# EPICS substitutions: llrfHlsAsynApp/Db/llrfHlsAsyn.substitutions
file config.db
{
    pattern {   DEVICE,  NELM_BL, NELM_HARMO  }
            {  "$(DEV)",    4096,         18  }
}

file status.db
{
    pattern {   DEVICE,  NELM_ALPHA  }
             { "$(DEV)",          7  }
}

file config_ch.db
{
    pattern { CH,  DEVICE   }
            {  0,  "$(DEV)" }
            {  1,  "$(DEV)" }
            {  2,  "$(DEV)" }
            {  3,  "$(DEV)" }
            {  4,  "$(DEV)" }
            {  5,  "$(DEV)" }
            {  6,  "$(DEV)" }
            {  7,  "$(DEV)" }
            {  8,  "$(DEV)" }
            {  9,  "$(DEV)" }
}

file config_ts.db
{
    pattern { TS, TS_N,  DEVICE  }
            {  0,   00, "$(DEV)" }
            {  1,   01, "$(DEV)" }
            {  2,   02, "$(DEV)" }
            {  3,   03, "$(DEV)" }
            {  4,   04, "$(DEV)" }
            {  5,   05, "$(DEV)" }
            {  6,   06, "$(DEV)" }
            {  7,   07, "$(DEV)" }
            {  8,   08, "$(DEV)" }
            {  9,   09, "$(DEV)" }
#
            { 10,   10, "$(DEV)" }
            { 11,   11, "$(DEV)" }
            { 12,   12, "$(DEV)" }
            { 13,   13, "$(DEV)" }
            { 14,   14, "$(DEV)" }
            { 15,   15, "$(DEV)" }
            { 16,   16, "$(DEV)" }
            { 17,   17, "$(DEV)" }
}

file status_ch.db
{
    pattern { CH, WND, DEVICE  }
            {  0,   0, "$(DEV)" }
            {  1,   0, "$(DEV)" }
            {  2,   0, "$(DEV)" }
            {  3,   0, "$(DEV)" }
            {  4,   0, "$(DEV)" }
            {  5,   0, "$(DEV)" }
            {  6,   0, "$(DEV)" }
            {  7,   0, "$(DEV)" }
            {  8,   0, "$(DEV)" }
            {  9,   0, "$(DEV)" }
#
            {  0,   1, "$(DEV)" }
            {  1,   1, "$(DEV)" }
            {  2,   1, "$(DEV)" }
            {  3,   1, "$(DEV)" }
            {  4,   1, "$(DEV)" }
            {  5,   1, "$(DEV)" }
            {  6,   1, "$(DEV)" }
            {  7,   1, "$(DEV)" }
            {  8,   1, "$(DEV)" }
            {  9,   1, "$(DEV)" }
#
            {  0,   2, "$(DEV)" }
            {  1,   2, "$(DEV)" }
            {  2,   2, "$(DEV)" }
            {  3,   2, "$(DEV)" }
            {  4,   2, "$(DEV)" }
            {  5,   2, "$(DEV)" }
            {  6,   2, "$(DEV)" }
            {  7,   2, "$(DEV)" }
            {  8,   2, "$(DEV)" }
            {  9,   2, "$(DEV)" }

}

file status_ts.db
{
    pattern { TS, TS_N,  DEVICE  }
            {  0,   00, "$(DEV)" }
            {  1,   01, "$(DEV)" }
            {  2,   02, "$(DEV)" }
            {  3,   03, "$(DEV)" }
            {  4,   04, "$(DEV)" }
            {  5,   05, "$(DEV)" }
            {  6,   06, "$(DEV)" }
            {  7,   07, "$(DEV)" }
            {  8,   08, "$(DEV)" }
            {  9,   09, "$(DEV)" }
#
            { 10,   10, "$(DEV)" }
            { 11,   11, "$(DEV)" }
            { 12,   12, "$(DEV)" }
            { 13,   13, "$(DEV)" }
            { 14,   14, "$(DEV)" }
            { 15,   15, "$(DEV)" }
            { 16,   16, "$(DEV)" }
            { 17,   17, "$(DEV)" }
}

file iq_wf_ch.db
{
    pattern { CH,  NELM,  DEVICE  }
            {  0,  4096, "$(DEV)" }
            {  1,  4096, "$(DEV)" }
            {  2,  4096, "$(DEV)" }
            {  3,  4096, "$(DEV)" }
            {  4,  4096, "$(DEV)" }
            {  5,  4096, "$(DEV)" }
            {  6,  4096, "$(DEV)" }
            {  7,  4096, "$(DEV)" }
            {  8,  4096, "$(DEV)" }
            {  9,  4096, "$(DEV)" }
}

file iq_wf_all.db
{
    pattern {  DEVICE  }
            { "$(DEV)" }
}

file avg_window.db
{
    pattern { NELM,  DEVICE,  WND  }
            { 4096, "$(DEV)",   0  }
            { 4096, "$(DEV)",   1  }
            { 4096, "$(DEV)",   2  }
}

file fastPV.db
{

    pattern { TS, TS_N,  DEVICE  }
            {  0,   00, "$(DEV)" }
            {  1,   01, "$(DEV)" }
            {  2,   02, "$(DEV)" }
            {  3,   03, "$(DEV)" }
            {  4,   04, "$(DEV)" }
            {  5,   05, "$(DEV)" }
            {  6,   06, "$(DEV)" }
            {  7,   07, "$(DEV)" }
            {  8,   08, "$(DEV)" }
            {  9,   09, "$(DEV)" }
#
            { 10,   10, "$(DEV)" }
            { 11,   11, "$(DEV)" }
            { 12,   12, "$(DEV)" }
            { 13,   13, "$(DEV)" }
            { 14,   14, "$(DEV)" }
            { 15,   15, "$(DEV)" }
            { 16,   16, "$(DEV)" }
            { 17,   17, "$(DEV)" }

}

file Bsa.db
{
  pattern {  DEVICE      ,  ATRB          , LNK      ,  EGU     ,  HOPR,  LOPR  }
          { "$(DEV):FB"  , "FAST_PACT"    , ""       , "degrees", "180", "-180" }
          { "$(DEV):FB"  , "FAST_AACT"    , ""       , "norm"   ,   "1",    "0" }
          { "$(DEV)"     , "BVOLT_PK_FAST", ""       , "kV"     ,    "",    "0" }
#
          {"$(DEV):W0C0" , "FAST_PACT"    , ""       , "degrees", "180", "-180" }
          {"$(DEV):W0C1" , "FAST_PACT"    , ""       , "degrees", "180", "-180" }
          {"$(DEV):W0C2" , "FAST_PACT"    , ""       , "degrees", "180", "-180" }
          {"$(DEV):W0C3" , "FAST_PACT"    , ""       , "degrees", "180", "-180" }
          {"$(DEV):W0C4" , "FAST_PACT"    , ""       , "degrees", "180", "-180" }
          {"$(DEV):W0C5" , "FAST_PACT"    , ""       , "degrees", "180", "-180" }
          {"$(DEV):W0C6" , "FAST_PACT"    , ""       , "degrees", "180", "-180" }
          {"$(DEV):W0C7" , "FAST_PACT"    , ""       , "degrees", "180", "-180" }
          {"$(DEV):W0C8" , "FAST_PACT"    , ""       , "degrees", "180", "-180" }
          {"$(DEV):W0C9" , "FAST_PACT"    , ""       , "degrees", "180", "-180" }
#
          {"$(DEV):W1C0" , "FAST_PACT"    , ""       , "degrees", "180", "-180" }
          {"$(DEV):W1C1" , "FAST_PACT"    , ""       , "degrees", "180", "-180" }
          {"$(DEV):W1C2" , "FAST_PACT"    , ""       , "degrees", "180", "-180" }
          {"$(DEV):W1C3" , "FAST_PACT"    , ""       , "degrees", "180", "-180" }
          {"$(DEV):W1C4" , "FAST_PACT"    , ""       , "degrees", "180", "-180" }
          {"$(DEV):W1C5" , "FAST_PACT"    , ""       , "degrees", "180", "-180" }
          {"$(DEV):W1C6" , "FAST_PACT"    , ""       , "degrees", "180", "-180" }
          {"$(DEV):W1C7" , "FAST_PACT"    , ""       , "degrees", "180", "-180" }
          {"$(DEV):W1C8" , "FAST_PACT"    , ""       , "degrees", "180", "-180" }
          {"$(DEV):W1C9" , "FAST_PACT"    , ""       , "degrees", "180", "-180" }
#
          {"$(DEV):W2C0" , "FAST_PACT"    , ""       , "degrees", "180", "-180" }
          {"$(DEV):W2C1" , "FAST_PACT"    , ""       , "degrees", "180", "-180" }
          {"$(DEV):W2C2" , "FAST_PACT"    , ""       , "degrees", "180", "-180" }
          {"$(DEV):W2C3" , "FAST_PACT"    , ""       , "degrees", "180", "-180" }
          {"$(DEV):W2C4" , "FAST_PACT"    , ""       , "degrees", "180", "-180" }
          {"$(DEV):W2C5" , "FAST_PACT"    , ""       , "degrees", "180", "-180" }
          {"$(DEV):W2C6" , "FAST_PACT"    , ""       , "degrees", "180", "-180" }
          {"$(DEV):W2C7" , "FAST_PACT"    , ""       , "degrees", "180", "-180" }
          {"$(DEV):W2C8" , "FAST_PACT"    , ""       , "degrees", "180", "-180" }
          {"$(DEV):W2C9" , "FAST_PACT"    , ""       , "degrees", "180", "-180" }
#
          { "$(DEV):W0C0", "FAST_AACT"    , ""       , "norm"   ,   "1",    "0" }
          { "$(DEV):W0C1", "FAST_AACT"    , ""       , "norm"   ,   "1",    "0" }
          { "$(DEV):W0C2", "FAST_AACT"    , ""       , "norm"   ,   "1",    "0" }
          { "$(DEV):W0C3", "FAST_AACT"    , ""       , "norm"   ,   "1",    "0" }
          { "$(DEV):W0C4", "FAST_AACT"    , ""       , "norm"   ,   "1",    "0" }
          { "$(DEV):W0C5", "FAST_AACT"    , ""       , "norm"   ,   "1",    "0" }
          { "$(DEV):W0C6", "FAST_AACT"    , ""       , "norm"   ,   "1",    "0" }
          { "$(DEV):W0C7", "FAST_AACT"    , ""       , "norm"   ,   "1",    "0" }
          { "$(DEV):W0C8", "FAST_AACT"    , ""       , "norm"   ,   "1",    "0" }
          { "$(DEV):W0C9", "FAST_AACT"    , ""       , "norm"   ,   "1",    "0" }
#
          { "$(DEV):W1C0", "FAST_AACT"    , ""       , "norm"   ,   "1",    "0" }
          { "$(DEV):W1C1", "FAST_AACT"    , ""       , "norm"   ,   "1",    "0" }
          { "$(DEV):W1C2", "FAST_AACT"    , ""       , "norm"   ,   "1",    "0" }
          { "$(DEV):W1C3", "FAST_AACT"    , ""       , "norm"   ,   "1",    "0" }
          { "$(DEV):W1C4", "FAST_AACT"    , ""       , "norm"   ,   "1",    "0" }
          { "$(DEV):W1C5", "FAST_AACT"    , ""       , "norm"   ,   "1",    "0" }
          { "$(DEV):W1C6", "FAST_AACT"    , ""       , "norm"   ,   "1",    "0" }
          { "$(DEV):W1C7", "FAST_AACT"    , ""       , "norm"   ,   "1",    "0" }
          { "$(DEV):W1C8", "FAST_AACT"    , ""       , "norm"   ,   "1",    "0" }
          { "$(DEV):W1C9", "FAST_AACT"    , ""       , "norm"   ,   "1",    "0" }
#
          { "$(DEV):W2C0", "FAST_AACT"    , ""       , "norm"   ,   "1",    "0" }
          { "$(DEV):W2C1", "FAST_AACT"    , ""       , "norm"   ,   "1",    "0" }
          { "$(DEV):W2C2", "FAST_AACT"    , ""       , "norm"   ,   "1",    "0" }
          { "$(DEV):W2C3", "FAST_AACT"    , ""       , "norm"   ,   "1",    "0" }
          { "$(DEV):W2C4", "FAST_AACT"    , ""       , "norm"   ,   "1",    "0" }
          { "$(DEV):W2C5", "FAST_AACT"    , ""       , "norm"   ,   "1",    "0" }
          { "$(DEV):W2C6", "FAST_AACT"    , ""       , "norm"   ,   "1",    "0" }
          { "$(DEV):W2C7", "FAST_AACT"    , ""       , "norm"   ,   "1",    "0" }
          { "$(DEV):W2C8", "FAST_AACT"    , ""       , "norm"   ,   "1",    "0" }
          { "$(DEV):W2C9", "FAST_AACT"    , ""       , "norm"   ,   "1",    "0" }
}

###########################
# PDES/ADES configuration #
###########################
file rfTSmux.db
{
    pattern {  DEVICE  }
            { "$(DEV)" }
}

####################
#Timing Abstraction#
####################

file cpswTimingCore.db
{
    pattern {   TRIG, TRIGMODE, CHANNEL,  DEVICE  }
            { "LLRF",  "ACCEL",   "00" , "$(DEV)" }
            { "LLRF",  "STDBY",   "01" , "$(DEV)" }
            {  "MOD",  "ACCEL",   "02" , "$(DEV)" }
            {  "MOD",  "STDBY",   "03" , "$(DEV)" }
            { "SSSB",  "ACCEL",   "04" , "$(DEV)" }
            { "SSSB",  "STDBY",   "05" , "$(DEV)" }
            {  "RTM",  "ACCEL",   "06" , "$(DEV)" }
            {  "RTM",  "STDBY",   "07" , "$(DEV)" }
           {"DAQMUX",  "ACCEL",   "08" , "$(DEV)" }
           {"DAQMUX",  "STDBY",   "09" , "$(DEV)" }
}

file cpswTimingCoreIndvDelay.db
{
    pattern {  TRIG ,  DEVICE  }
            { "LLRF", "$(DEV)" }
            {  "MOD", "$(DEV)" }
            { "SSSB", "$(DEV)" }
            {  "RTM", "$(DEV)" }
           {"DAQMUX", "$(DEV)" }
}

file cpswTimingCoreDelay.db
{
    pattern {  DEVICE  }
            { "$(DEV)" }
}

file waveformTimeAxis.db
{
    pattern {   DEVICE  , DESC                         ,  SIZE ,  FREQ   }
            {  "$(DEV)" , "HLS waveform time axis"     , "4096" , "357"  }
}
